Fanuc KAREL source: ke00004.KL

-- PROVISIONAL review KL for V940-1; original PC SHA256 58d631a4fedb51eea196d238300f53162e513dad9ddef2d76a1dc313f848e2e8
-- Incomplete behavior may be omitted. Consult companion uncertainty JSON. Do not deploy.
PROGRAM KE00004
%NOLOCKGROUP
BEGIN
  -- V9_ZERO_TABLE_METADATA_HINT layout=0002_ascii; no indexed target words; source/name/runtime held
  -- UNRESOLVED_PC offsets 5-12; opcodes 9D,23
  -- UNRESOLVED_PC offsets 17-29; opcodes 3F,75
  -- UNRESOLVED_PC offsets 34-58; opcodes 27,22,22,2A,22,31
  -- UNRESOLVED_PC offsets 63-67; opcodes 7F
END KE00004
